// TIA Portal V19 export
TYPE "LEXCHANGETRAY_typeRollerVfdContronNodeCommands"
// vfdSportsIncEnable: Bool
// vfdSportsIncReset: Bool
// sinaCommands: LBC_typeSinaSpeedControlNodeCommands
// stored: Access Published
   STRUCT
      vfdSportsIncEnable : Bool;
      vfdSportsIncReset : Bool;
      sinaCommands : "LBC_typeSinaSpeedControlNodeCommands";
   END_STRUCT;
END_TYPE
